(*
Abstract base block for periodic signal generators.

Provides :attr:`Period`, :attr:`Amplitude`, :attr:`Bias`, and :attr:`Phase`
as shared properties for all periodic signal generators. Derived blocks can
implement :meth:`Run` and :meth:`Reset` to produce their specific waveform.

.. note::
   Direct calls to this function block are not permitted (``no_explicit_call``).
   Extend it and call the derived block instead.
*)
{attribute 'enable_dynamic_creation'}
{attribute 'no_explicit_call' := 'direct call for this function block is not allowed'}
FUNCTION_BLOCK ABSTRACT FB_PeriodicSignal EXTENDS FB_SoComponent
IMPLEMENTS I_PeriodicSignal
VAR
	_tPeriod    : LTIME; // Duration of one full cycle. Must be greater than zero.
	_fAmplitude : LREAL; // Scales the raw wave. Output swings between Bias ± Amplitude.
	_fBias      : LREAL; // Shifts the output vertically.
	_fPhase     : LREAL; // Phase offset in radians. Shifts the wave horizontally.
END_VAR

(*
Gets or sets the amplitude. 

The output swings between ``Bias + Amplitude`` and ``Bias - Amplitude``.
*)
PROPERTY Amplitude : LREAL
GET
Amplitude := THIS^._fAmplitude;
END_GET
SET
THIS^._fAmplitude := Amplitude;
END_SET
END_PROPERTY

(*
Gets or sets the bias.

This is a fixed offset added to the output, shifting the wave up or down.
*)
PROPERTY Bias : LREAL
GET
Bias := THIS^._fBias;
END_GET
SET
THIS^._fBias := Bias;
END_SET
END_PROPERTY

(* 
Gets or sets the period. 

This is the time taken to complete one full cycle.
*)
PROPERTY Period : LTIME
GET
Period := THIS^._tPeriod;
END_GET
SET
THIS^._tPeriod := Period;
END_SET
END_PROPERTY

(*
Gets or sets the phase offset in radians.

This shifts the wave horizontally. Negative values shift in the opposite direction.
*)
PROPERTY Phase : LREAL
GET
Phase := THIS^._fPhase;
END_GET
SET
THIS^._fPhase := Phase;
END_SET
END_PROPERTY

END_FUNCTION_BLOCK

(* stored: Version 1.1.0.1, ProductVersion 3.1.4024.15
   POU FB_PeriodicSignal: Id {cbd39e12-2ae0-475d-bc34-310fd8fb240c}, SpecialFunc None
   Property Amplitude: Id {e33b959c-5507-4fe5-8252-6648d80eb04e}
   Get Get: Id {3187b26c-6eec-4705-b7df-8dfd98e2a0e0}
   Set Set: Id {0380e645-9c7c-4297-9818-1fbfb667941c}
   Property Bias: Id {cf70a9ab-678a-4268-8982-5635b0e4b580}
   Get Get: Id {dcbbafb7-395e-494b-847a-d5612c4c1269}
   Set Set: Id {9afdc719-4056-4f16-a4d8-b3979882453e}
   Property Period: Id {6589787f-fa06-4b3f-a6b3-cb90872faddb}
   Get Get: Id {a9ca5ea3-b5f5-476a-ac0d-bb3ecf0e2701}
   Set Set: Id {013e4795-3451-4f4b-9236-9a7f593eda5a}
   Property Phase: Id {6ccd7cf2-c9c6-4976-b356-fb63aac7f16d}
   Get Get: Id {0928e42b-1ed4-4159-943b-8d54041ae22f}
   Set Set: Id {50f6b25e-aa59-4efa-a1cc-2e14b65a1de4} *)
